// SIMATIC S7-200 SMART project (STEP 7-Micro/WIN SMART), CPU SR20

SYMBOL_TABLE 风机和阀
温度量程下限           VD232
温度量程上限           VD228
模拟量最大值           VD216
模拟量最小值           VD208
压力量程下限           VD252
压力量程上限           VD268
风机停止             V2.0
风机启动             V2.1
风机远程             V2.2
风机故障             V2.4
风机输出             V2.5
风机               V2.6
阀1停止             V2.7
阀1启动             V3.0
阀1远程             V3.1
阀1故障             V3.2
阀1输出             V3.3
阀1               V5.6
阀2停止             V3.4
阀2启动             V3.5
阀2远程             V3.6
阀2故障             V3.7
阀2输出             V4.0
阀2               V4.1
阀3停止             V4.2
阀3启动             V4.3
阀3远程             V4.4
阀3故障             V4.5
阀3输出             V4.6
阀3               V4.7
阀4停止             V5.0
阀4启动             V5.1
阀4远程             V5.2
阀4故障             V5.3
阀4输出             V5.4
阀4               V5.5
END_SYMBOL_TABLE

SYMBOL_TABLE 系统符号
Always_On        SM0.0    // 始终接通
END_SYMBOL_TABLE

SYMBOL_TABLE 点火烧嘴
点火命令1            M0.0
点火成功信号1          M0.1
故障复位1            M1.3     // 输出
点火变压器1           M1.0     // 输出
点火电磁阀1           M1.1     // 输出
报警1              M1.2     // 输出
点火命令2            M0.2
点火成功信号2          M0.3
故障复位2            M1.4     // 输出
点火变压器2           M1.5     // 输出
点火电磁阀2           M1.6     // 输出
报警2              M1.7     // 输出
END_SYMBOL_TABLE

ORGANIZATION_BLOCK MAIN:OB1
TITLE=程序注释
BEGIN
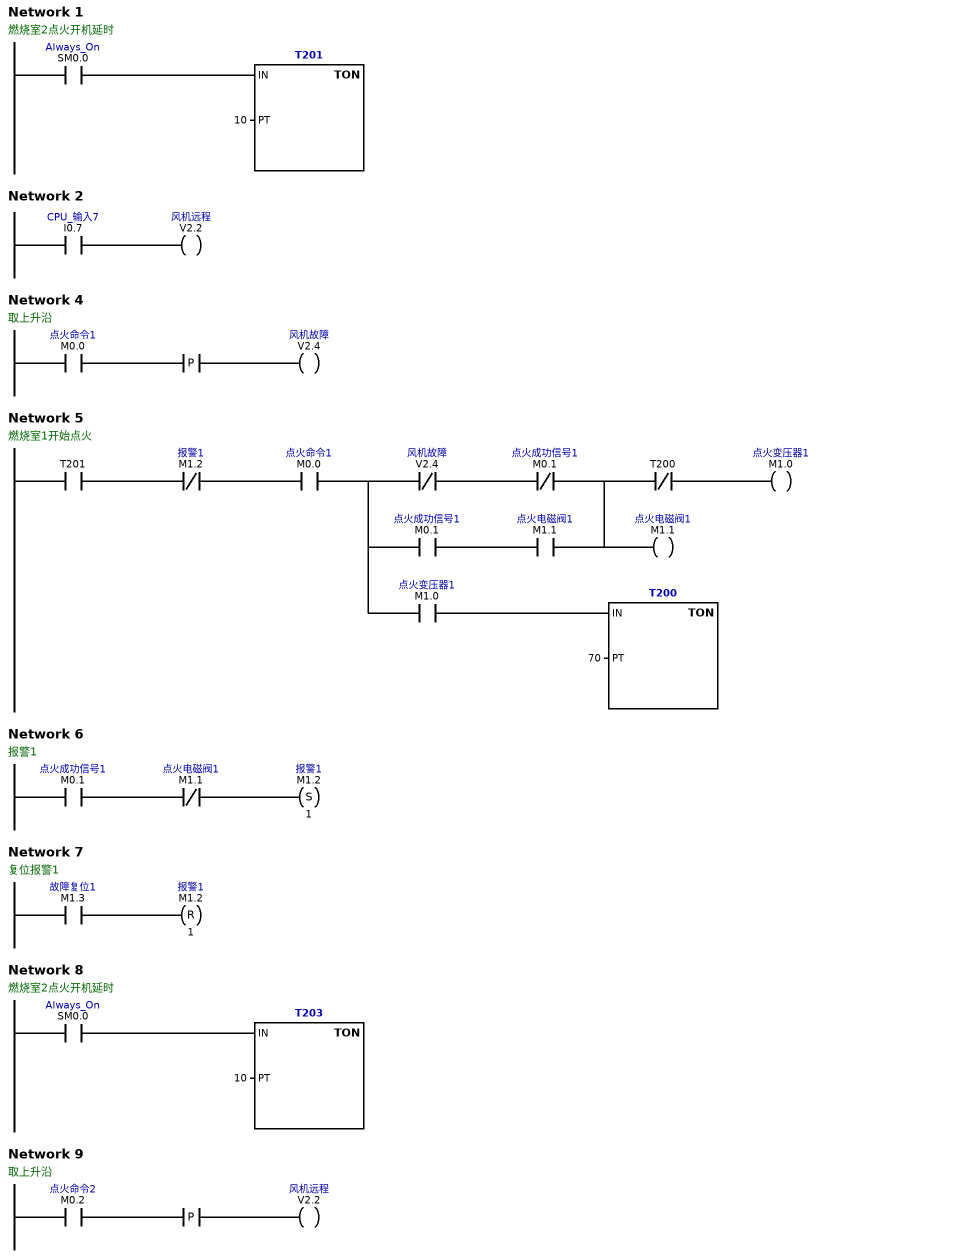
Network 1
// 燃烧室2点火开机延时
LD     Always_On:SM0.0
TON    T201, 10
Network 2
LD     CPU_输入7:I0.7
=      风机远程:V2.2
Network 4
// 取上升沿
LD     点火命令1:M0.0
EU
=      风机故障:V2.4
Network 5
// 燃烧室1开始点火
// (network saved uncompiled; LAD cells follow)
// row 0: c0 -| |- T201  c1 -|/|- 报警1:M1.2  c2 -| |- 点火命令1:M0.0 v  c3 -|/|- 风机故障:V2.4  c4 -|/|- 点火成功信号1:M0.1 v  c5 -|/|- T200  c6 -( ) 点火变压器1:M1.0
// row 1: c2 ^v  c3 -| |- 点火成功信号1:M0.1  c4 -| |- 点火电磁阀1:M1.1 ^  c5 -( ) 点火电磁阀1:M1.1
// row 2: c2 ^  c3 -| |- 点火变压器1:M1.0  c4 --  c5 [TON T200 IN:=power@row2, PT:=70]
// row 3: c5 [box]
Network 6
// 报警1
LD     点火成功信号1:M0.1
AN     点火电磁阀1:M1.1
S      报警1:M1.2, 1
Network 7
// 复位报警1
LD     故障复位1:M1.3
R      报警1:M1.2, 1
Network 8
// 燃烧室2点火开机延时
LD     Always_On:SM0.0
TON    T203, 10
Network 9
// 取上升沿
LD     点火命令2:M0.2
EU
=      风机远程:V2.2
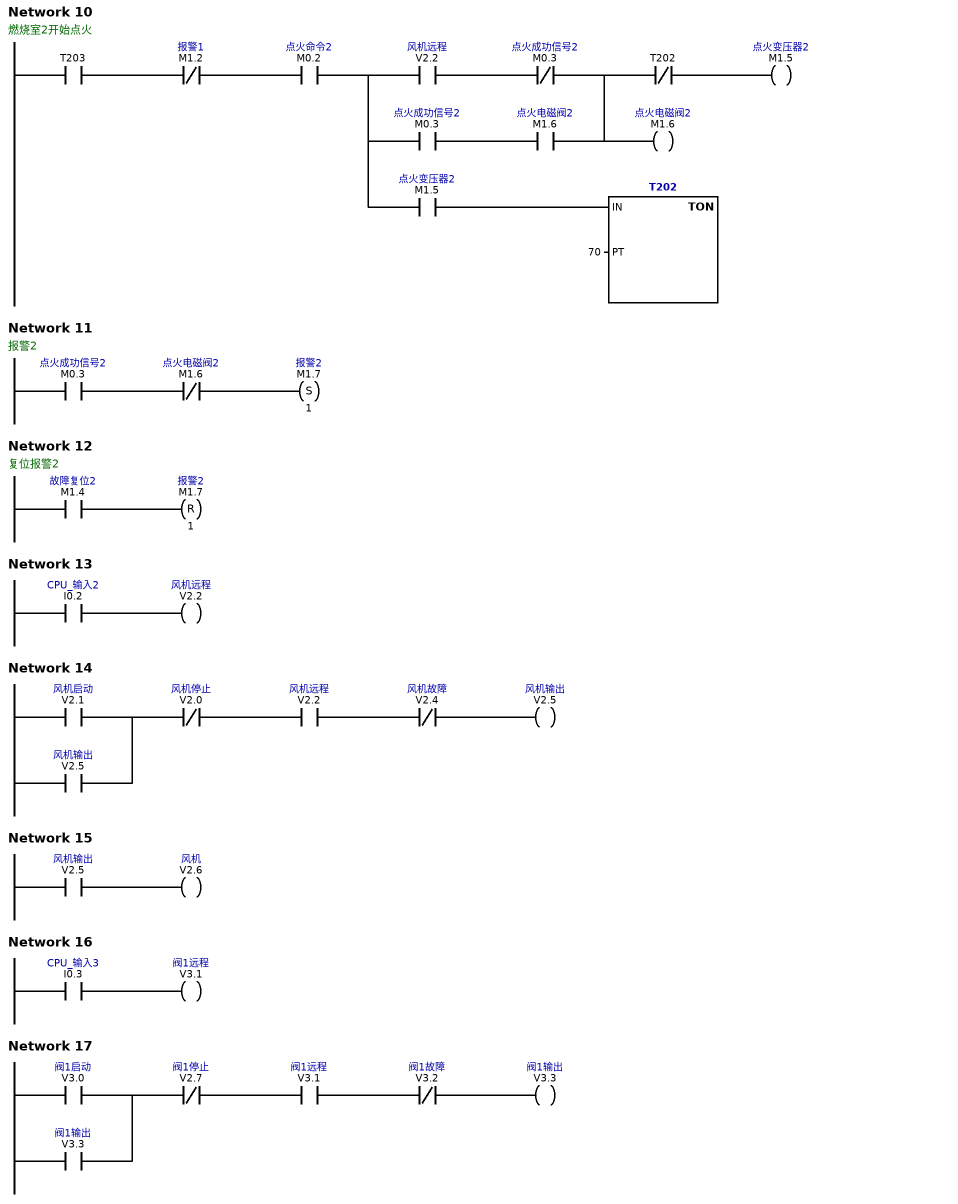
Network 10
// 燃烧室2开始点火
LD     T203
AN     报警1:M1.2
A      点火命令2:M0.2
LPS
LD     风机远程:V2.2
AN     点火成功信号2:M0.3
LD     点火成功信号2:M0.3
A      点火电磁阀2:M1.6
OLD
ALD
LPS
AN     T202
=      点火变压器2:M1.5
LPP
=      点火电磁阀2:M1.6
LPP
A      点火变压器2:M1.5
TON    T202, 70
Network 11
// 报警2
LD     点火成功信号2:M0.3
AN     点火电磁阀2:M1.6
S      报警2:M1.7, 1
Network 12
// 复位报警2
LD     故障复位2:M1.4
R      报警2:M1.7, 1
Network 13
LD     CPU_输入2:I0.2
=      风机远程:V2.2
Network 14
LD     风机启动:V2.1
O      风机输出:V2.5
AN     风机停止:V2.0
A      风机远程:V2.2
AN     风机故障:V2.4
=      风机输出:V2.5
Network 15
LD     风机输出:V2.5
=      风机:V2.6
Network 16
// (network saved uncompiled; LAD cells follow)
// row 0: c0 -| |- CPU_输入3:I0.3  c1 -( ) 阀1远程:V3.1
Network 17
// (network saved uncompiled; LAD cells follow)
// row 0: c0 -| |- 阀1启动:V3.0 v  c1 -|/|- 阀1停止:V2.7  c2 -| |- 阀1远程:V3.1  c3 -|/|- 阀1故障:V3.2  c4 -( ) 阀1输出:V3.3
// row 1: c0 -| |- 阀1输出:V3.3 ^
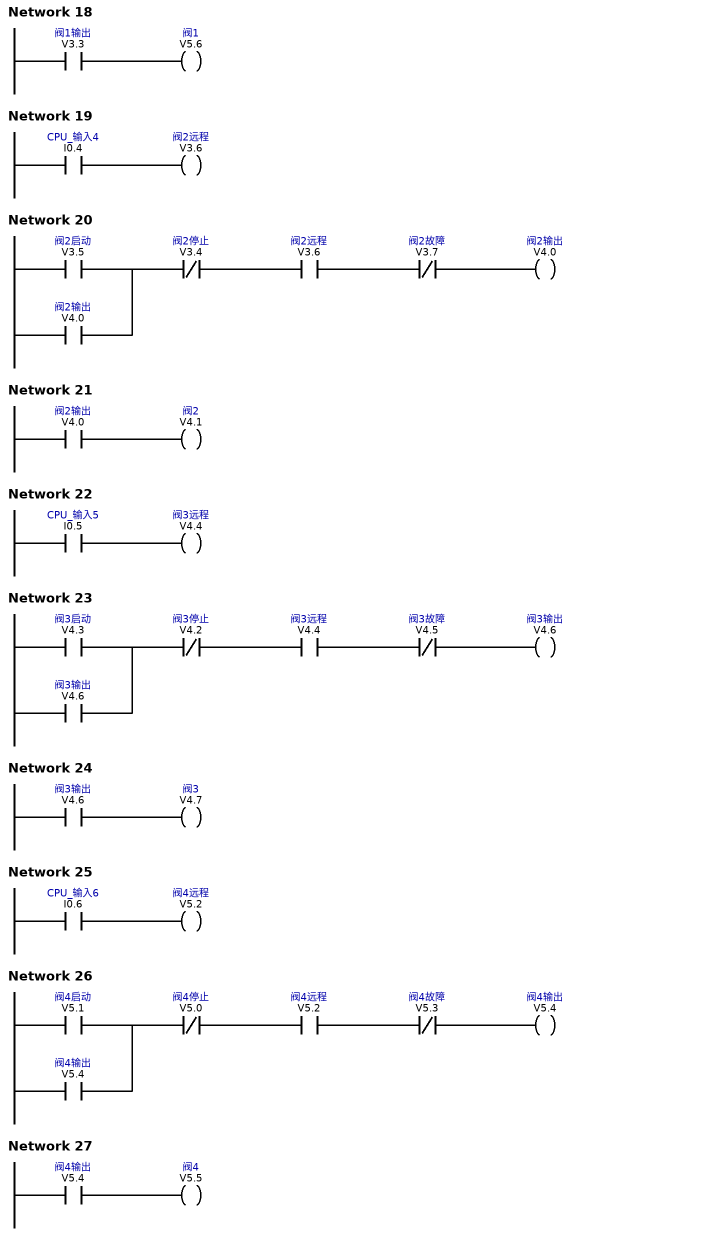
Network 18
// (network saved uncompiled; LAD cells follow)
// row 0: c0 -| |- 阀1输出:V3.3  c1 -( ) 阀1:V5.6
Network 19
// (network saved uncompiled; LAD cells follow)
// row 0: c0 -| |- CPU_输入4:I0.4  c1 -( ) 阀2远程:V3.6
Network 20
// (network saved uncompiled; LAD cells follow)
// row 0: c0 -| |- 阀2启动:V3.5 v  c1 -|/|- 阀2停止:V3.4  c2 -| |- 阀2远程:V3.6  c3 -|/|- 阀2故障:V3.7  c4 -( ) 阀2输出:V4.0
// row 1: c0 -| |- 阀2输出:V4.0 ^
Network 21
// (network saved uncompiled; LAD cells follow)
// row 0: c0 -| |- 阀2输出:V4.0  c1 -( ) 阀2:V4.1
Network 22
LD     CPU_输入5:I0.5
=      阀3远程:V4.4
Network 23
LD     阀3启动:V4.3
O      阀3输出:V4.6
AN     阀3停止:V4.2
A      阀3远程:V4.4
AN     阀3故障:V4.5
=      阀3输出:V4.6
Network 24
LD     阀3输出:V4.6
=      阀3:V4.7
Network 25
LD     CPU_输入6:I0.6
=      阀4远程:V5.2
Network 26
LD     阀4启动:V5.1
O      阀4输出:V5.4
AN     阀4停止:V5.0
A      阀4远程:V5.2
AN     阀4故障:V5.3
=      阀4输出:V5.4
Network 27
LD     阀4输出:V5.4
=      阀4:V5.5
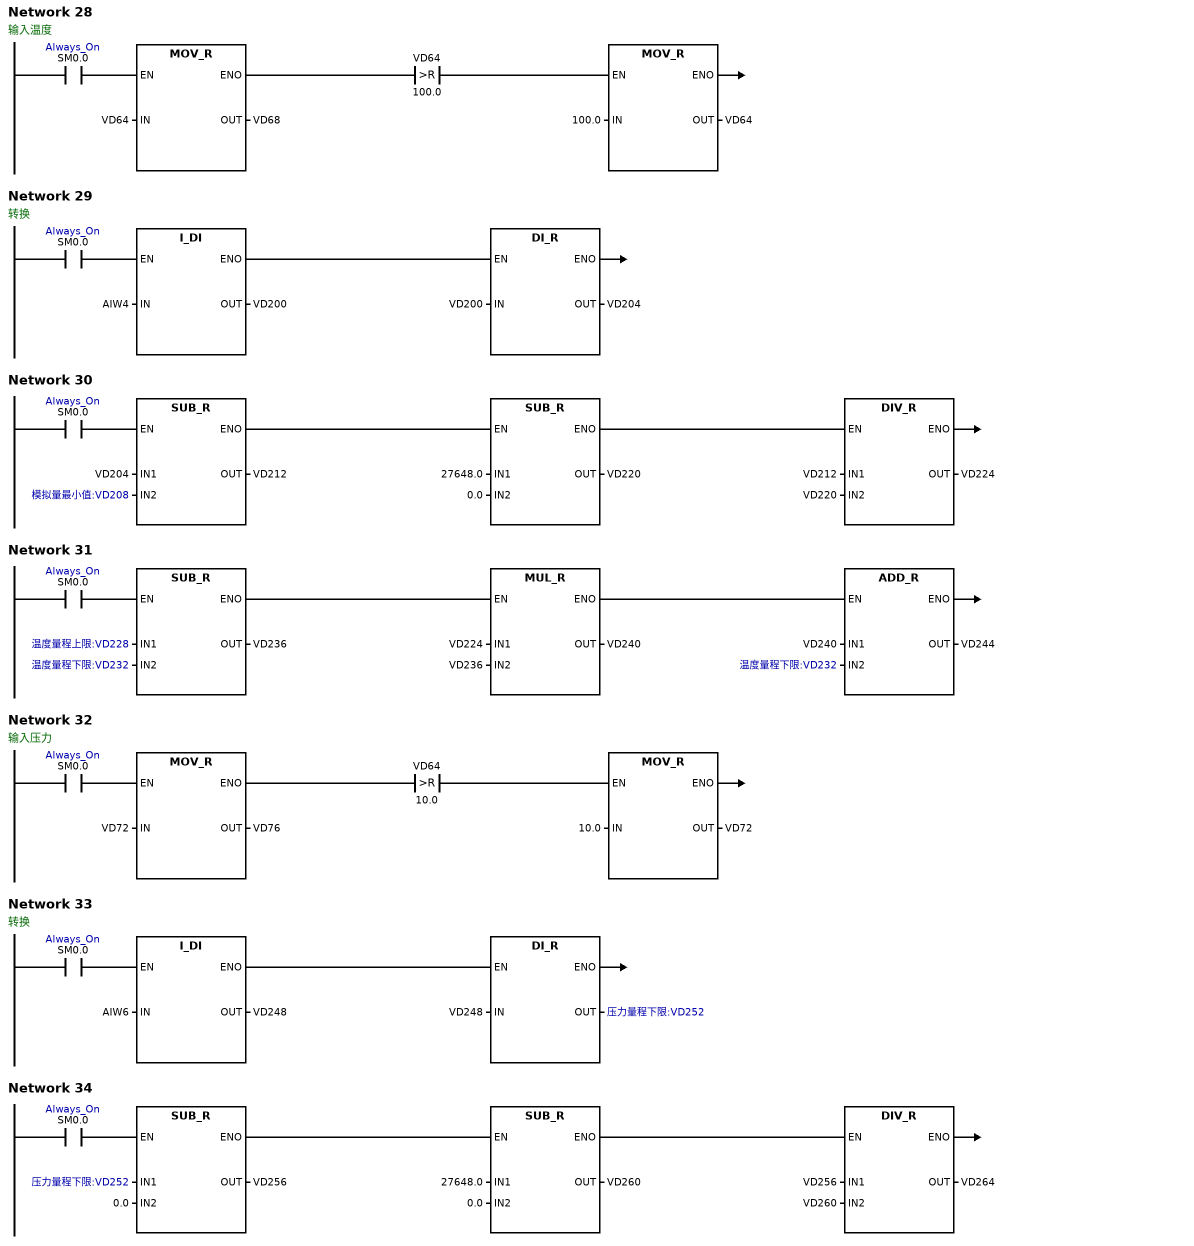
Network 28
// 输入温度
// (network saved uncompiled; LAD cells follow)
// row 0: c0 -| |- Always_On:SM0.0  c1 [MOV_R EN:=power@row0, IN:=VD64, ENO=>power, OUT=>VD68]  c2 --  c3 -|>R|- VD64, 100.0  c4 --  c5 [MOV_R EN:=power@row0, IN:=100.0, ENO=>power, OUT=>VD64]  c6 ->
// row 1: c1 [box]  c5 [box]
Network 29
// 转换
// (network saved uncompiled; LAD cells follow)
// row 0: c0 -| |- Always_On:SM0.0  c1 [I_DI EN:=power@row0, IN:=AIW4, ENO=>power, OUT=>VD200]  c2 --  c3 --  c4 [DI_R EN:=power@row0, IN:=VD200, ENO=>power, OUT=>VD204]  c5 ->
// row 1: c1 [box]  c4 [box]
Network 30
// (network saved uncompiled; LAD cells follow)
// row 0: c0 -| |- Always_On:SM0.0  c1 [SUB_R EN:=power@row0, IN1:=VD204, IN2:=模拟量最小值:VD208, ENO=>power, OUT=>VD212]  c2 --  c3 --  c4 [SUB_R EN:=power@row0, IN1:=27648.0, IN2:=0.0, ENO=>power, OUT=>VD220]  c5 --  c6 --  c7 [DIV_R EN:=power@row0, IN1:=VD212, IN2:=VD220, ENO=>power, OUT=>VD224]  c8 ->
// row 1: c1 [box]  c4 [box]  c7 [box]
Network 31
// (network saved uncompiled; LAD cells follow)
// row 0: c0 -| |- Always_On:SM0.0  c1 [SUB_R EN:=power@row0, IN1:=温度量程上限:VD228, IN2:=温度量程下限:VD232, ENO=>power, OUT=>VD236]  c2 --  c3 --  c4 [MUL_R EN:=power@row0, IN1:=VD224, IN2:=VD236, ENO=>power, OUT=>VD240]  c5 --  c6 --  c7 [ADD_R EN:=power@row0, IN1:=VD240, IN2:=温度量程下限:VD232, ENO=>power, OUT=>VD244]  c8 ->
// row 1: c1 [box]  c4 [box]  c7 [box]
Network 32
// 输入压力
// (network saved uncompiled; LAD cells follow)
// row 0: c0 -| |- Always_On:SM0.0  c1 [MOV_R EN:=power@row0, IN:=VD72, ENO=>power, OUT=>VD76]  c2 --  c3 -|>R|- VD64, 10.0  c4 --  c5 [MOV_R EN:=power@row0, IN:=10.0, ENO=>power, OUT=>VD72]  c6 ->
// row 1: c1 [box]  c5 [box]
Network 33
// 转换
// (network saved uncompiled; LAD cells follow)
// row 0: c0 -| |- Always_On:SM0.0  c1 [I_DI EN:=power@row0, IN:=AIW6, ENO=>power, OUT=>VD248]  c2 --  c3 --  c4 [DI_R EN:=power@row0, IN:=VD248, ENO=>power, OUT=>压力量程下限:VD252]  c5 ->
// row 1: c1 [box]  c4 [box]
Network 34
// (network saved uncompiled; LAD cells follow)
// row 0: c0 -| |- Always_On:SM0.0  c1 [SUB_R EN:=power@row0, IN1:=压力量程下限:VD252, IN2:=0.0, ENO=>power, OUT=>VD256]  c2 --  c3 --  c4 [SUB_R EN:=power@row0, IN1:=27648.0, IN2:=0.0, ENO=>power, OUT=>VD260]  c5 --  c6 --  c7 [DIV_R EN:=power@row0, IN1:=VD256, IN2:=VD260, ENO=>power, OUT=>VD264]  c8 ->
// row 1: c1 [box]  c4 [box]  c7 [box]
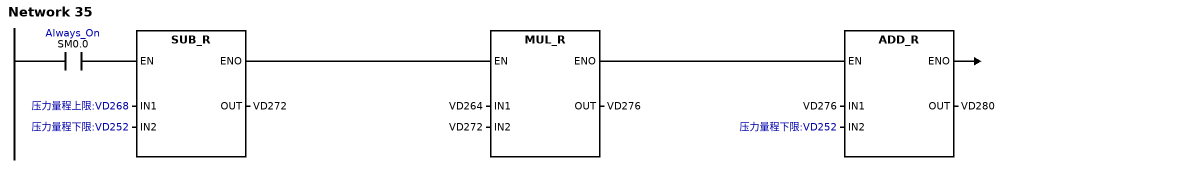
Network 35
// (network saved uncompiled; LAD cells follow)
// row 0: c0 -| |- Always_On:SM0.0  c1 [SUB_R EN:=power@row0, IN1:=压力量程上限:VD268, IN2:=压力量程下限:VD252, ENO=>power, OUT=>VD272]  c2 --  c3 --  c4 [MUL_R EN:=power@row0, IN1:=VD264, IN2:=VD272, ENO=>power, OUT=>VD276]  c5 --  c6 --  c7 [ADD_R EN:=power@row0, IN1:=VD276, IN2:=压力量程下限:VD252, ENO=>power, OUT=>VD280]  c8 ->
// row 1: c1 [box]  c4 [box]  c7 [box]
END_ORGANIZATION_BLOCK

// SBR1: protected block, not included

// SBR2: protected block, not included

// SBR3: protected block, not included

// SBR4: protected block, not included

// SBR5: protected block, not included

// SBR6: protected block, not included

// SBR7: protected block, not included
